// TIA Portal V21 program export: 0 tag tables, 0 data types, 1 data blocks, 2 code blocks (in call order from the OBs), 0 instance data blocks

DATA_BLOCK "TempoCiclo"   // DB1
{ S7_Optimized_Access := 'TRUE' }
// stored: MemoryReserve 100
   VAR
      TempoEsecuzioneSezioni : Array[0.."K_NumKTipo"] of Struct
         Actual : LReal;
         Appo : LReal;
         Perc : Real;
      END_STRUCT;
      TempoEsecuzioneTotale : LReal := 58.6982355555555;
   END_VAR
BEGIN
   TempoEsecuzioneSezioni[0].Actual := 59.6303733333333;
   TempoEsecuzioneSezioni[1].Actual := 10.6522622222222;
   TempoEsecuzioneSezioni[2].Actual := 2.87701333333333;
   TempoEsecuzioneSezioni[3].Actual := 0.0813733333333333;
   TempoEsecuzioneSezioni[4].Actual := 0.0;
   TempoEsecuzioneSezioni[5].Actual := 0.122457777777778;
   TempoEsecuzioneSezioni[6].Actual := 9.52839555555556;
   TempoEsecuzioneSezioni[7].Actual := 0.0;
   TempoEsecuzioneSezioni[8].Actual := 30.8047644444444;
   TempoEsecuzioneSezioni[9].Actual := 0.0;
   TempoEsecuzioneSezioni[10].Actual := 1.09750222222222;
   TempoEsecuzioneSezioni[11].Actual := 1.80765777777778;
   TempoEsecuzioneSezioni[12].Actual := 1.59227111111111;
   TempoEsecuzioneSezioni[13].Actual := 0.335724444444444;
   TempoEsecuzioneSezioni[14..15].Actual := 0.0;
   TempoEsecuzioneSezioni[16].Actual := 0.411697777777778;
   TempoEsecuzioneSezioni[0].Appo := 16#0002_CA53_756E_9C20;
   TempoEsecuzioneSezioni[1].Appo := 16#0002_CA53_7425_DC42;
   TempoEsecuzioneSezioni[2].Appo := 16#0002_CA53_7439_A22C;
   TempoEsecuzioneSezioni[3].Appo := 16#0002_CA53_743A_5594;
   TempoEsecuzioneSezioni[4].Appo := 0.0;
   TempoEsecuzioneSezioni[5].Appo := 16#0002_CA53_747C_A09E;
   TempoEsecuzioneSezioni[6].Appo := 16#0002_CA53_747B_C4C4;
   TempoEsecuzioneSezioni[7].Appo := 0.0;
   TempoEsecuzioneSezioni[8].Appo := 16#0002_CA53_7550_3BFC;
   TempoEsecuzioneSezioni[9].Appo := 0.0;
   TempoEsecuzioneSezioni[10].Appo := 16#0002_CA53_7576_EA36;
   TempoEsecuzioneSezioni[11].Appo := 16#0002_CA53_7566_5B52;
   TempoEsecuzioneSezioni[12].Appo := 16#0002_CA53_7577_EA3C;
   TempoEsecuzioneSezioni[13].Appo := 16#0002_CA53_7559_EF26;
   TempoEsecuzioneSezioni[14..15].Appo := 0.0;
   TempoEsecuzioneSezioni[16].Appo := 16#0002_CA53_7553_6340;
   TempoEsecuzioneSezioni[0].Perc := 101.588;
   TempoEsecuzioneSezioni[1].Perc := 18.1475;
   TempoEsecuzioneSezioni[2].Perc := 4.901362;
   TempoEsecuzioneSezioni[3].Perc := 0.1386299;
   TempoEsecuzioneSezioni[4].Perc := 0.0;
   TempoEsecuzioneSezioni[5].Perc := 0.2086226;
   TempoEsecuzioneSezioni[6].Perc := 16.23285;
   TempoEsecuzioneSezioni[7].Perc := 0.0;
   TempoEsecuzioneSezioni[8].Perc := 52.47988;
   TempoEsecuzioneSezioni[9].Perc := 0.0;
   TempoEsecuzioneSezioni[10].Perc := 0.8256088;
   TempoEsecuzioneSezioni[11].Perc := 3.079578;
   TempoEsecuzioneSezioni[12].Perc := 2.712639;
   TempoEsecuzioneSezioni[13].Perc := 0.5719498;
   TempoEsecuzioneSezioni[14..15].Perc := 0.0;
   TempoEsecuzioneSezioni[16].Perc := 0.7013801;
   // TempoEsecuzioneSezioni[1] : Analogica
   // TempoEsecuzioneSezioni[2] : Pid
   // TempoEsecuzioneSezioni[3] : Portata
   // TempoEsecuzioneSezioni[4] : Trend
   // TempoEsecuzioneSezioni[5] : Paratia
   // TempoEsecuzioneSezioni[6] : Motore
   // TempoEsecuzioneSezioni[7] : Allarme
   // TempoEsecuzioneSezioni[8] : Valvola
   // TempoEsecuzioneSezioni[9] : SezionePastorizzatore
   // TempoEsecuzioneSezioni[10] : Zona
   // TempoEsecuzioneSezioni[11] : Comunicazione
   // TempoEsecuzioneSezioni[12] : Sequenza
   // TempoEsecuzioneSezioni[13] : SegnaliMacchine
   // TempoEsecuzioneSezioni[14] : Sensore
   // TempoEsecuzioneSezioni[15] : Additivo
   // TempoEsecuzioneSezioni[16] : Ricetta
END_DATA_BLOCK

ORGANIZATION_BLOCK "Main Richiamo"   // OB1, LAD, ProgramCycle
TITLE = "Main Program Sweep (Cycle)"
{ S7_Optimized_Access := 'TRUE' }
// stored: SetENOAutomatically false
   VAR_INPUT
      Initial_Call : Bool;
      Remanence : Bool;
   END_VAR
   VAR_TEMP
      TempoEsecuzione : LReal;
      TempoEsecuzioneTotale : LReal;
      "Counter" : Int;
      AppoTemp : DInt;
   END_VAR
BEGIN

REGION Network 1 (SCL)
   #TempoEsecuzione := RUNTIME("TempoCiclo".TempoEsecuzioneSezioni[0].Appo) * 1000.0;
   REGION Richiamo base software
       "GestDatiUtili"();

       IF "K_NumZona" > 0 THEN
           #TempoEsecuzione := RUNTIME("TempoCiclo".TempoEsecuzioneSezioni[K_TipoZona].Appo) * 1000.0;
           "Main zone"();
           "TempoCiclo".TempoEsecuzioneSezioni[K_TipoZona].Actual := RUNTIME("TempoCiclo".TempoEsecuzioneSezioni[K_TipoZona].Appo) * 1000.0;
       END_IF;


       "LogoCliente".K_LogoCliente_1 := "K_LogoCliente_Brain";
       "LogoCliente".K_LogoCliente_2 := "K_LogoCliente_Dubit";

       // "LogoCliente".K_LogoCliente_1 := "K_LogoCliente_Brain";
       // "LogoCliente".K_LogoCliente_2 := "K_LogoCliente_Greci";

       //"GestTema"();
       //"GestLogin"();
       //"GestScreensaver"();
   END_REGION ;
   REGION 0040 Sequenze
       IF "K_NumSequenza" > 0 THEN
           #TempoEsecuzione := RUNTIME("TempoCiclo".TempoEsecuzioneSezioni[K_TipoSequenza].Appo) * 1000.0;
           "Main sequenze"();
           "TempoCiclo".TempoEsecuzioneSezioni[K_TipoSequenza].Actual := RUNTIME("TempoCiclo".TempoEsecuzioneSezioni[K_TipoSequenza].Appo) * 1000.0;
       END_IF;
   END_REGION ;
   REGION 0060 Strumentazione
       IF "K_NumAnalogica" > 0 THEN
           #TempoEsecuzione := RUNTIME("TempoCiclo".TempoEsecuzioneSezioni[K_TipoAnalogica].Appo) * 1000.0;
           "Main analogiche"();
           "TempoCiclo".TempoEsecuzioneSezioni[K_TipoAnalogica].Actual := RUNTIME("TempoCiclo".TempoEsecuzioneSezioni[K_TipoAnalogica].Appo) * 1000.0;
       END_IF;
       IF "K_NumPid" > 0 THEN
           #TempoEsecuzione := RUNTIME("TempoCiclo".TempoEsecuzioneSezioni[K_TipoPid].Appo) * 1000.0;
           "Main pid"();
           "TempoCiclo".TempoEsecuzioneSezioni[K_TipoPid].Actual := RUNTIME("TempoCiclo".TempoEsecuzioneSezioni[K_TipoPid].Appo) * 1000.0;
       END_IF;
       IF "K_NumPortata" > 0 THEN
           #TempoEsecuzione := RUNTIME("TempoCiclo".TempoEsecuzioneSezioni[K_TipoPortata].Appo) * 1000.0;
           "Main Portate"();
           "TempoCiclo".TempoEsecuzioneSezioni[K_TipoPortata].Actual := RUNTIME("TempoCiclo".TempoEsecuzioneSezioni[K_TipoPortata].Appo) * 1000.0;
       END_IF;
       IF "K_NumTrends" > 0 THEN
           #TempoEsecuzione := RUNTIME("TempoCiclo".TempoEsecuzioneSezioni[K_TipoTrend].Appo) * 1000.0;
           "Main trends"();
           "TempoCiclo".TempoEsecuzioneSezioni[K_TipoTrend].Actual := RUNTIME("TempoCiclo".TempoEsecuzioneSezioni[K_TipoTrend].Appo) * 1000.0;
       END_IF;
       IF "K_NumStazione" > 1 THEN
           "Main instradatore"();
       END_IF;
   END_REGION ;
   REGION 0070 Utenze/Attuatori
       IF "K_NumMotore" > 0 THEN
           #TempoEsecuzione := RUNTIME("TempoCiclo".TempoEsecuzioneSezioni[K_TipoMotore].Appo) * 1000.0;
           "Main motori"();
           "TempoCiclo".TempoEsecuzioneSezioni[K_TipoMotore].Actual := RUNTIME("TempoCiclo".TempoEsecuzioneSezioni[K_TipoMotore].Appo) * 1000.0;
       END_IF;
       IF "K_NumParatia" > 0 THEN
           #TempoEsecuzione := RUNTIME("TempoCiclo".TempoEsecuzioneSezioni[K_TipoParatia].Appo) * 1000.0;
           "Main paratie"();
           "TempoCiclo".TempoEsecuzioneSezioni[K_TipoParatia].Actual := RUNTIME("TempoCiclo".TempoEsecuzioneSezioni[K_TipoParatia].Appo) * 1000.0;
       END_IF;
       IF "K_NumValvola" > 0 THEN
           #TempoEsecuzione := RUNTIME("TempoCiclo".TempoEsecuzioneSezioni[K_TipoValvola].Appo) * 1000.0;
           "Main valvole"();
           "TempoCiclo".TempoEsecuzioneSezioni[K_TipoValvola].Actual := RUNTIME("TempoCiclo".TempoEsecuzioneSezioni[K_TipoValvola].Appo) * 1000.0;
       END_IF;
   END_REGION
   REGION 0090 Ricette
       IF "K_NumMacchinaARicetta" > 0 THEN
           #TempoEsecuzione := RUNTIME("TempoCiclo".TempoEsecuzioneSezioni[K_TipoRicetta].Appo) * 1000.0;
           "Main ricette"();
           "TempoCiclo".TempoEsecuzioneSezioni[K_TipoRicetta].Actual := RUNTIME("TempoCiclo".TempoEsecuzioneSezioni[K_TipoRicetta].Appo) * 1000.0;
       END_IF;
   END_REGION ;
   REGION Macchinari
       "GestioneMacchina_010102"();
   END_REGION ;
   REGION 8000 Segnali macchina
       IF "K_NumSegnaleMacchina" > 0 THEN
           #TempoEsecuzione := RUNTIME("TempoCiclo".TempoEsecuzioneSezioni[K_TipoSegnaliMacchine].Appo) * 1000.0;
           "Main SegnaliMacchina"();
           "TempoCiclo".TempoEsecuzioneSezioni[K_TipoSegnaliMacchine].Actual := RUNTIME("TempoCiclo".TempoEsecuzioneSezioni[K_TipoSegnaliMacchine].Appo) * 1000.0;
       END_IF;
   END_REGION ;
   REGION 9000 Comunicazione
       IF "K_NumComunicazioneS7" > 0 THEN
           #TempoEsecuzione := RUNTIME("TempoCiclo".TempoEsecuzioneSezioni[K_TipoComunicazione].Appo) * 1000.0;
           "GetPut"();
           "TempoCiclo".TempoEsecuzioneSezioni[K_TipoComunicazione].Actual := RUNTIME("TempoCiclo".TempoEsecuzioneSezioni[K_TipoComunicazione].Appo) * 1000.0;
       END_IF;
   END_REGION ;
   "TempoCiclo".TempoEsecuzioneSezioni[0].Actual := RUNTIME("TempoCiclo".TempoEsecuzioneSezioni[0].Appo) * 1000.0;
   REGION Esecuzione totale
       REGION CalcoloTempoEsecuzioneTotale
           #TempoEsecuzioneTotale := 0;
           FOR #Counter := 1 TO "K_NumKTipo" DO
               #TempoEsecuzioneTotale += "TempoCiclo".TempoEsecuzioneSezioni[#Counter].Actual;
           END_FOR;
           "TempoCiclo".TempoEsecuzioneTotale := #TempoEsecuzioneTotale;
       END_REGION ;
       REGION Calcolo percentuale di incisione percentuale
           FOR #Counter := 0 TO "K_NumKTipo" DO
               "TempoCiclo".TempoEsecuzioneSezioni[#Counter].Perc := LREAL_TO_REAL("TempoCiclo".TempoEsecuzioneSezioni[#Counter].Actual / "TempoCiclo".TempoEsecuzioneTotale * 100.0);
           END_FOR;
       END_REGION ;
   END_REGION ;
END_REGION
END_ORGANIZATION_BLOCK

ORGANIZATION_BLOCK "Main Richiamo Pid"   // OB35, LAD, CyclicInterrupt
TITLE = "Cyclic Interrupt"
{ S7_Optimized_Access := 'FALSE' }
// stored: AutoNumber false, SetENOAutomatically false
   VAR_TEMP
      OB35_EV_CLASS : Byte;   // Bits 0-3 = 1 (Coming event), Bits 4-7 = 1 (Event class 1)
      OB35_STRT_INF : Byte;   // 16#36 (OB 35 has started)
      OB35_PRIORITY : Byte;   // 11 (Priority of 1 is lowest)
      OB35_OB_NUMBR : Byte;   // 35 (Organization block 35, OB35)
      OB35_RESERVED_1 : Byte;   // Reserved for system
      OB35_RESERVED_2 : Byte;   // Reserved for system
      OB35_PHASE_OFFSET : Word;   // Phase offset (msec)
      OB35_RESERVED_3 : Int;   // Reserved for system
      OB35_EXC_FREQ : Int;   // Frequency of execution (msec)
      OB35_DATE_TIME : Date_And_Time;   // Date and time OB35 started
      LMN_ABS : Real;
      Appo : Real;
      FLD_ACT_ENG : Real;
      Appo_PID : Real;
      Appo_OUT : Real;
      Reset : Bool;
      PEW : Word;
      PAW : Int;
      OUT_INT : Int;
      OUT_REAL : Real;
      MinLimit : Bool;
      MaxLimit : Bool;
      "Appo Pew pid4" : Word;
      SogliaImpostataCorrettamente : Bool;
      DA_inserire : "Std_VarGestAnalog";
      VelrichiestaMotore : Int;
   END_VAR
   VAR CONSTANT
      Isteresi : Int;
   END_VAR
BEGIN

REGION Network 1 (SCL): CALL PID
   "Pid_Sterilizzatore_Pompamono"();
   "Pid_Sterilizzatore_Pompapistoni"();
   "Pid_Sterilizzatore_RaffreddamentoAcqua"();
   "Pid_Sterilizzatore_RiscaldamentoAcqua"();
   "Pid_Sterilizzatore_RiscaldamentoProdotto"();
END_REGION
END_ORGANIZATION_BLOCK
